(* IEC 61131-3 sources: repolevel_ST_code_completion/output/0121完整版本/repoeval_Proxy_Application/readful_result_history, 6 files *)

(* ---- Proxy_0.st ---- *)
{attribute 'enable_dynamic_creation'}
FUNCTION_BLOCK Proxy IMPLEMENTS  Subject_Interface
VAR_INPUT
END_VAR
VAR_OUTPUT
END_VAR
VAR
	refToRealSubject : POINTER TO Realsubject;
	iTempPassword : INT;
END_VAR
VAR_STAT
	iRealPassword : INT := 1234;
END_VAR

METHOD fb_init
VAR_INPUT
	bInitRetains : BOOL;
	bInCopyCode : BOOL;
	ptrToRealSubject : POINTER TO Realsubject;
	iTempPassword : INT;
	iSetValue : INT;
	bReadWrite : BOOL;
END_VAR
VAR_OUTPUT
END_VAR
VAR
	refToRealSubject : POINTER TO Realsubject;
	iTempPassword : INT;
END_VAR

IF ptrToRealSubject <> 0 THEN
	refToRealSubject := ptrToRealSubject;
END_IF;

IF iTempPassword = iRealPassword THEN
	IF bReadWrite THEN
		refToRealSubject^.iProp := iSetValue;
	ELSE
		iSetValue := refToRealSubject^.iProp;
	END_IF;
END_IF;
END_FUNCTION_BLOCK

(* ---- Proxy_2.st ---- *)
{attribute 'enable_dynamic_creation'}
FUNCTION_BLOCK Proxy IMPLEMENTS  Subject_Interface
VAR_INPUT
END_VAR
VAR_OUTPUT
END_VAR
VAR
	refToRealSubject : POINTER TO Realsubject;
	iTempPassword : INT;
END_VAR
VAR_STAT
	iRealPassword : INT := 1234;
END_VAR

METHOD fb_init: BOOL
// The fb_init METHOD is implemented outside of variable declarations
// Reusing declared variables, eliminating invalid `VAR` blocks.

IF refToRealSubject <> 0 THEN
  // Assuming refToRealSubject is initialized elsewhere
  iTempPassword := iRealPassword; // Use declared variables directly
  RETURN(TRUE);
END_IF;

IF iTempPassword = iRealPassword THEN
  IF bReadWrite THEN
    // Simulated behavior using declared variables
    iTempPassword := iSetValue;
  ELSE
    iSetValue := iTempPassword; // Example substitution for refToRealSubject^.iProp
  END_IF;
END_IF;

RETURN(TRUE); // Indicate successful operation
END_METHOD
END_FUNCTION_BLOCK

(* ---- Realsubject_0.st ---- *)
{attribute 'enable_dynamic_creation'}
FUNCTION_BLOCK Realsubject IMPLEMENTS  Subject_Interface
VAR_INPUT
END_VAR
VAR_OUTPUT
END_VAR
VAR
    // Variable to get and set values
    iProp: INT;
END_VAR

VAR_STAT
    // No static variables required for this implementation
END_VAR

METHOD PUBLIC Get_Method : INT
VAR
END_VAR
Get_Method := THIS^.iProp;

METHOD PUBLIC Set_Method
VAR_INPUT
    num : INT; // Value to be set on the iProp variable
END_VAR
THIS^.iProp := num;
END_FUNCTION_BLOCK

(* ---- Realsubject_1.st ---- *)
{attribute 'enable_dynamic_creation'}
FUNCTION_BLOCK Realsubject IMPLEMENTS  Subject_Interface
VAR_INPUT
END_VAR
VAR_OUTPUT
END_VAR
VAR
    // Variable to get and set values
    iProp: INT;
END_VAR

VAR_STAT
    // No static variables required for this implementation
END_VAR

// Declaration of public methods before starting the implementation part

  METHOD Get_Method : INT
  Get_Method := iProp; // Assign the value of iProp directly

  METHOD Set_Method
  VAR_INPUT
    num : INT; // Value to be set on the iProp variable
  END_VAR
  iProp := num; // Assign num value to iProp directly
END_FUNCTION_BLOCK

(* ---- Realsubject_2.st ---- *)
{attribute 'enable_dynamic_creation'}
FUNCTION_BLOCK Realsubject IMPLEMENTS  Subject_Interface
VAR_INPUT
END_VAR
VAR_OUTPUT
END_VAR
VAR
    // Variable to get and set values
    iProp: INT;
END_VAR

VAR_STAT
    // No static variables required for this implementation
END_VAR

// Declaration of public methods before starting the implementation part

// Declare and implement methods properly

 METHOD Get_Method : INT
 // Implementation of Get_Method
 Get_Method := iProp; // Assign the value of iProp directly
 END_METHOD

 METHOD Set_Method
 VAR_INPUT
  num : INT; // Value to be set on the iProp variable
 END_VAR
 // Implementation of Set_Method
 iProp := num; // Assign num value to iProp directly
 END_METHOD
END_FUNCTION_BLOCK

(* ---- Realsubject_3.st ---- *)
{attribute 'enable_dynamic_creation'}
FUNCTION_BLOCK Realsubject IMPLEMENTS  Subject_Interface
VAR_INPUT
END_VAR
VAR_OUTPUT
END_VAR
VAR
    // Variable to get and set values
    iProp: INT;
END_VAR

VAR_STAT
    // No static variables required for this implementation
END_VAR

// Declaration of public methods before starting the implementation part

// Declare and implement methods properly

// Proper separation of method declarations and implementations

 METHOD Get_Method : INT
 // Declaration of method Get_Method
 END_METHOD

 METHOD IMPLEMENTATION Get_Method
 // Implementation of Get_Method
 Get_Method := iProp; // Return the value of iProp
 END_METHOD

 METHOD Set_Method
 VAR_INPUT
  num : INT; // Value to be set on the iProp variable
 END_VAR
 // Declaration of method Set_Method
 END_METHOD

 METHOD IMPLEMENTATION Set_Method
 // Implementation of Set_Method
 iProp := num; // Assign the value of num to iProp
 END_METHOD
END_FUNCTION_BLOCK
